FUNCTION_BLOCK FB_Regelingen_1
VAR
	internalBesturingsMode : E_Besturingsmodus;
	internalRegelschuifStandV2013 : SINT;
	internalRegelschuifStandV2022 : SINT;
	internalToerentalP2011 : INT;
	internalToerentalP2021 : INT;
END_VAR

internalToerentalP2011 := 50;
internalToerentalP2021 := 70;

PROPERTY BestuurMode : E_Besturingsmodus
GET
BestuurMode := internalBesturingsMode;
END_GET
SET
internalBesturingsMode := BestuurMode ;
END_SET
END_PROPERTY

PROPERTY RegelschuifStandV2013 : SINT
GET
RegelschuifStandV2013 := internalRegelschuifStandV2013;
END_GET
SET
internalRegelschuifStandV2013 := RegelschuifStandV2013;
END_SET
END_PROPERTY

PROPERTY RegelschuifStandV2022 : SINT
GET
RegelschuifStandV2022 := internalRegelschuifStandV2022;
END_GET
SET
internalRegelschuifStandV2022 := RegelschuifStandV2022;
END_SET
END_PROPERTY

PROPERTY ToerentalP2011 : INT
GET
ToerentalP2011 := internalToerentalP2011;
END_GET
SET
internalToerentalP2011 := ToerentalP2011;
END_SET
END_PROPERTY

PROPERTY ToerentalP2021 : INT
GET
ToerentalP2011 := internalToerentalP2021;
END_GET
SET
internalToerentalP2011 := ToerentalP2021;
END_SET
END_PROPERTY

END_FUNCTION_BLOCK

(* stored: Version 1.1.0.1, ProductVersion 3.1.4026.8
   POU FB_Regelingen_1: Id {ba4530f9-bec4-46f8-8992-3ba5eead477b}, SpecialFunc None
   Folder Properties: Id {7c6e2fb9-4775-4dab-baa7-e5b89aec5c3b}
   Property BestuurMode: Id {ef2a99b5-5f20-4b0a-b6bc-351e2bd448d2}
   Get Get: Id {e2d7c206-8f7f-426b-82b2-78ed55082002}
   Set Set: Id {8657565b-1ccc-48a7-a1b2-ee5eec85ab16}
   Property RegelschuifStandV2013: Id {22aaed06-7a4e-4fb5-9a38-f497238e5600}
   Get Get: Id {df927b81-0b19-4ba5-8491-c549fdf3679f}
   Set Set: Id {46201dd7-77e4-4f26-9ef1-8e4e09797119}
   Property RegelschuifStandV2022: Id {25ca217c-5af0-4a23-9400-b185b560c6f4}
   Get Get: Id {baefb7a1-259b-4e50-b712-7341c25b1805}
   Set Set: Id {9059e5f4-2721-43bc-8e0e-724abee52b74}
   Property ToerentalP2011: Id {a0f08cbb-fea4-4e47-9c72-4a53599b6c38}
   Get Get: Id {cde78827-a38d-4b92-81d4-9333a5eb2ad4}
   Set Set: Id {c50b0b11-1f65-436f-bc39-0a87e0b63fbe}
   Property ToerentalP2021: Id {8985ff52-3298-4fc8-aa83-ceecf5a234e2}
   Get Get: Id {64ce7207-5106-4e28-8d0f-a19017054c1e}
   Set Set: Id {810193cf-b8f4-44af-854a-e5e0ee173417} *)
